SUBAPPLICATION Uebung_026_sub (* Spiegelabfolge (6) *)
  (* Standard: 61499-2; Description: Copyright (c) 2024 Meisterschulen am Ostbahnhof This program and the accompanying materials are made available under the terms of the Eclipse Public License 2.0 which is available at https://www.eclipse.org/legal/epl-2.0/ SPDX-License-Identifier: EPL-2.0 *)
  (* Version 1.0, 2024-02-05, Franz Höpfinger, Meisterschulen am Ostbahnhof *)
  IMPORT logiBUS::io::DQ::logiBUS_DO;
  IMPORT logiBUS::io::DQ::logiBUS_DO_S;
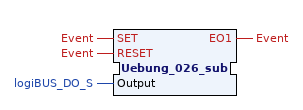
  EVENT_INPUT
    SET;
    RESET;
  END_EVENT
  EVENT_OUTPUT
    EO1;
  END_EVENT
  VAR_INPUT
    Output : logiBUS::io::DQ::logiBUS_DO_S := logiBUS_DO::Invalid; (* Identify the Output Output_Q1..Q8 *)
  END_VAR
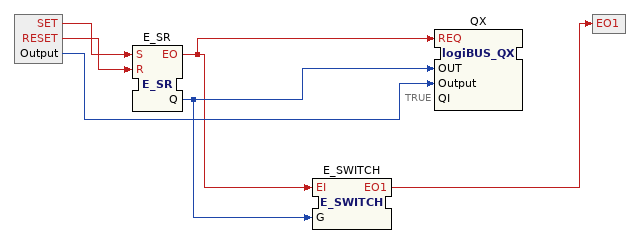
  FBS
    E_SR : iec61499::events::E_SR;
    QX : logiBUS::io::DQ::logiBUS_QX(QI := TRUE);
    E_SWITCH : iec61499::events::E_SWITCH;
  END_FBS
  EVENT_CONNECTIONS
    E_SR.EO TO QX.REQ;
    E_SR.EO TO E_SWITCH.EI;
    SET TO E_SR.S;
    RESET TO E_SR.R;
    E_SWITCH.EO1 TO EO1;
  END_CONNECTIONS
  DATA_CONNECTIONS
    E_SR.Q TO QX.OUT;
    E_SR.Q TO E_SWITCH.G;
    Output TO QX.Output;
  END_CONNECTIONS
END_SUBAPPLICATION
